FUNCTION_BLOCK FB_HwRefNanotecPD EXTENDS FB_CanNodeBase
VAR_INPUT
	nControlword	AT%Q* : UINT;
	nMode			AT%Q* : SINT;
	nTargetPosition AT%Q* : DINT;
	nTargetSpeed	AT%Q* : INT;
	nDriveSubMode	AT%Q* : UDINT; //1 für Move, 8 für Stillstand mit Stromabsenkung	
END_VAR
VAR_OUTPUT
	nStatusword 	 	AT%I* : UINT;
	nCurrentMode 	 	AT%I* : SINT;
	nCurrentPosition 	AT%I* : DINT;
	nCurrentSpeed		AT%I* : INT;
	nFollowingError		AT%I* : DINT;	
END_VAR
VAR
	bIsHomed 				: BOOL;
	eCurrentSTM				: E_CoDS402States;
	nState 					: USINT;
	bFirstTimeInOperational : BOOL := TRUE;
	
	nStateA_ProcessError	: USINT;
	nLastErrorID			: DWORD;
	nErrorCount				: USINT;
	
	nStateA_ResetError		: USINT;
END_VAR

VAR PERSISTENT
	nDistPerMotorRev	: DINT;
	nRefPos				: DINT;
	nHomePos			: DINT;
	nSlowHomingSpeed	: DINT;
	nFastHomingSpeed	: DINT;
	bInvertInitDir		: BOOL;
	nMinPos				: DINT;
	nMaxPos				: DINT;
	nMaxSpeed			: DINT;
END_VAR

//In der Basisklasse wird A_Prepare und A_ResetApp ausgeführt
//ResetApp ist hier nicht relevant.

eCurrentSTM := M_GetDS402State();
CASE nState OF
	0:	//Prepare
		SUPER^();
		IF bPreparingOK THEN
			nState := 1;
		END_IF
		
	1:	//Operational
		//Wenn hier zum erstem mal hineingesprungen wird, und in error, dann gleich resetten
		IF eCurrentSTM = E_CoDS402States.DS402STATE_Fault OR eCurrentSTM = E_CoDS402States.DS402STATE_FaultReactionActive THEN
			IF bFirstTimeInOperational THEN
				nState := 4;
			ELSE
				nState := 2;
			END_IF
		END_IF
		bFirstTimeInOperational := FALSE;
		
	2:	//Process error
		A_ProcessError();
		IF nStateA_ProcessError = 80 THEN
			//Error auswerten - es werden nur die untersten 16Bit ausgewertet (Error Code siehe Doku NanoTec)
			nLastErrorID := nLastErrorID AND 16#FFFF;
			CASE nLastErrorID OF
				16#1000:	nErrorID := E_ErrorIdHwGeneral.ERRORID_GenericError;
				16#2300:	nErrorID := E_ErrorIdHwGeneral.ERRORID_MotorCurrentExceeded;
				16#3100:	nErrorID := E_ErrorIdHwGeneral.ERRORID_InvalidInputVoltage;
				16#4200:	nErrorID := E_ErrorIdHwGeneral.ERRORID_ControllerTemperature;
				16#5540:	nErrorID := E_ErrorIdHwGeneral.ERRORID_InterlockError;
				16#6010:	nErrorID := E_ErrorIdHwGeneral.ERRORID_SoftwareReset;
				16#6100:	nErrorID := E_ErrorIdHwGeneral.ERRORID_InternalSoftwareError;
				16#6320:	nErrorID := E_ErrorIdHwGeneral.ERRORID_InvalidRatedCurrent;
				16#7113:	nErrorID := E_ErrorIdHwGeneral.ERRORID_BallastResistorOverloaded;
				16#7121:	nErrorID := E_ErrorIdHwGeneral.ERRORID_MotorBlocked;
				16#7200:	nErrorID := E_ErrorIdHwGeneral.ERRORID_InternalError;
				16#7305:	nErrorID := E_ErrorIdHwGeneral.ERRORID_Sensor1Fault;
				16#7306:	nErrorID := E_ErrorIdHwGeneral.ERRORID_Sensor2Fault;
				16#7307:	nErrorID := E_ErrorIdHwGeneral.ERRORID_SensorNFault;
				16#7600:	nErrorID := E_ErrorIdHwGeneral.ERRORID_MemoryError;
				16#8000,16#8100: nErrorID := E_ErrorIdHwGeneral.ERRORID_FieldbusMonitoring;
				16#8130, 16#8200, 16#8210, 16#8220, 16#8240 : nErrorID := E_ErrorIdHwGeneral.ERRORID_CANopenError;	
				16#8400:	nErrorID := E_ErrorIdHwGeneral.ERRORID_SpeedMonitoring;
				16#8611:	nErrorID := E_ErrorIdHwGeneral.ERRORID_FollowingError;
				16#8612:	nErrorID := E_ErrorIdHwGeneral.ERRORID_LimitSwitchExceeded;
			ELSE
				nErrorID := 0;
			END_CASE
			nStateA_ProcessError := 0;
			//Notify error
			stError.HardwareGrp := stHardwareId.eGroup;
			stError.HardwareNr := stHardwareId.nItem;
			stError.POU := E_POU.POU_FB_HwRefNanotecPD;
			stError.POUAction := E_POUACT.POUACT_UNDEFIEND;
			stError.ErrorId := nErrorID;
			fbErrorList.M_Add(stError);
			nState := 3;
		END_IF
		
	3:	//Error
		IF bResetError THEN
			nState:= 4;
			bResetError := FALSE;
		END_IF
		bIsHomed := FALSE;
		bError := TRUE;
		
	4:	//Reset
		bBusy := TRUE;
		A_ResetError();
		IF nStateA_ResetError = 80 THEN
			bError := FALSE;
			bBusy := FALSE;
			nStateA_ResetError := 0;
			nState := 1;
		ELSIF nStateA_ResetError = 99 THEN
			bBusy := FALSE;
			nStateA_ResetError := 0;
			nState := 3;
		END_IF
	
END_CASE

ACTION A_ProcessError:
IF nStateA_ProcessError = 0 THEN
	//Object 0x1003:00 auslesen (Anzahl der Errors im Pre-defined error field)
	fbSdoRead(nIndex:= 16#1003, nSubIndex:= 0, nDataLength:= 1, bExecute:= TRUE);
	nErrorCount := 0;
	IF NOT fbSdoRead.bBusy THEN
		IF NOT fbSdoRead.bError THEN
			nErrorCount := DINT_TO_USINT(fbSdoRead.nData);
		END_IF
		fbSdoRead(bExecute:= FALSE);
		IF nErrorCount > 0 THEN
			nStateA_ProcessError := 1;
		ELSE
			nStateA_ProcessError := 80;
		END_IF
	END_IF
END_IF


IF nStateA_ProcessError = 1 THEN
	//Object 0x1003:01 auslesen (Neuester Error)
	fbSdoRead(nIndex:= 16#1003, nSubIndex:= 1, nDataLength:= 4, bExecute:= TRUE);
	nLastErrorID := 0;
	IF NOT fbSdoRead.bBusy THEN
		IF NOT fbSdoRead.bError THEN
			nLastErrorID := fbSdoRead.nData;
		END_IF
		fbSdoRead(bExecute:= FALSE);
		nStateA_ProcessError := 80;
	END_IF
END_IF
END_ACTION

ACTION A_ResetError:
CASE nStateA_ResetError OF
	0:	
		CASE eCurrentSTM OF
			E_CoDS402States.DS402STATE_Fault:
				nControlword := 153;	//Reset error
			E_CoDS402States.DS402STATE_SwitchOnDisabled:
				nStateA_ResetError := 1;
			E_CoDS402States.DS402STATE_ReadyToSwitchOn:
				nControlword := 0;	//Transition 7 in DS402 statemachine -> geht in Switch on disabled
				nStateA_ResetError := 1;
			E_CoDS402States.DS402STATE_SwitchedOn:
				nControlword := 0;	//Transition 10 in DS402 statemachine -> geht in Switch on disabled
				nStateA_ResetError := 1;
			E_CoDS402States.DS402STATE_OperationEnabled:
				nControlword := 0;	//Shutdown
				nStateA_ResetError := 1;
			E_CoDS402States.DS402STATE_NotReadyToSwitchOn:	//Statusword wahrscheinlich nicht gemappt
				nStateA_ResetError := 99;
		END_CASE
		
	1:	//Würde Antrieb bereits gehomed?
		IF bIsHomed THEN
			nControlword := 6;
			nStateA_ResetError := 2;
		ELSE
			nStateA_ResetError := 80;
		END_IF
		
	2:	IF eCurrentSTM = E_CoDS402States.DS402STATE_ReadyToSwitchOn THEN
			nControlword := 7;	//Change to "Switched on"
			nStateA_ResetError := 3;
		ELSIF eCurrentSTM = E_CoDS402States.DS402STATE_Fault THEN
			nStateA_ResetError := 99;
		END_IF
	
	3:	IF eCurrentSTM = E_CoDS402States.DS402STATE_SwitchedOn THEN
			nControlword := 15;	//Change to "Switched on"
			nStateA_ResetError := 4;
		ELSIF eCurrentSTM = E_CoDS402States.DS402STATE_Fault THEN
			nStateA_ResetError := 99;
		END_IF
		
	4:	IF eCurrentSTM = E_CoDS402States.DS402STATE_OperationEnabled THEN
			nStateA_ResetError := 80;
		ELSIF eCurrentSTM = E_CoDS402States.DS402STATE_Fault THEN
			nStateA_ResetError := 99;
		END_IF		
	
END_CASE
END_ACTION

METHOD M_GetDS402State : E_CoDS402States
VAR_INPUT
END_VAR
IF (nStatusword AND 16#4F) = 0 THEN
	M_GetDS402State := E_CoDS402States.DS402STATE_NotReadyToSwitchOn;
ELSIF (nStatusword AND 16#4F) = 16#40 THEN
	M_GetDS402State := E_CoDS402States.DS402STATE_SwitchOnDisabled;
ELSIF (nStatusword AND 16#6F) = 16#21 THEN
	M_GetDS402State := E_CoDS402States.DS402STATE_ReadyToSwitchOn;
ELSIF (nStatusword AND 16#6F) = 16#23 THEN
	M_GetDS402State := E_CoDS402States.DS402STATE_SwitchedOn;
ELSIF (nStatusword AND 16#6F) = 16#27 THEN
	M_GetDS402State := E_CoDS402States.DS402STATE_OperationEnabled;
ELSIF (nStatusword AND 16#6F) = 16#07 THEN
	M_GetDS402State := E_CoDS402States.DS402STATE_QuickStopActive;
ELSIF (nStatusword AND 16#4F) = 16#0F THEN
	M_GetDS402State := E_CoDS402States.DS402STATE_FaultReactionActive;
ELSIF (nStatusword AND 16#4F) = 16#08 THEN
	M_GetDS402State := E_CoDS402States.DS402STATE_Fault;
ELSE
	M_GetDS402State := E_CoDS402States.DS402STATE_Notspecified;
END_IF
END_METHOD

METHOD M_GetHomingState : E_CoDS402HomingState
VAR_INPUT
END_VAR

VAR 
END_VAR
//werted nur die Bits 10,12,13 vom Statusword aus
CASE nStatusword AND 16#3400 OF
	16#0000:	M_GetHomingState := E_CoDS402HomingState.HomingInProgress;
	16#0400:	M_GetHomingState := E_CoDS402HomingState.HomingInteruptedOrNotReached;
	16#1000:	M_GetHomingState := E_CoDS402HomingState.HomingAttainedButNotReached;
	16#1400:	M_GetHomingState := E_CoDS402HomingState.HomingSuccess;
	16#2000,
	16#2400		:M_GetHomingState := E_CoDS402HomingState.HomingError;
END_CASE
END_METHOD

METHOD M_RealToInternPos : DINT
VAR_INPUT
	nValue : DINT;
END_VAR
M_RealToInternPos := REAL_TO_DINT(DINT_TO_REAL(nValue) * 2000.0 / DINT_TO_REAL(nDistPerMotorRev));
END_METHOD

METHOD M_RealToInternSpeed : INT
VAR_INPUT
	nValue : DINT; //Speed in µm/s oder 1/100°/sec
END_VAR
//Umrechnung in U/min
M_RealToInternSpeed := REAL_TO_INT(DINT_TO_REAL(nValue) / DINT_TO_REAL(nDistPerMotorRev) * 60.0);
RETURN;
END_METHOD

METHOD M_SetTargetPos : BOOL
VAR_INPUT
	nValue : DINT; //Reale Einheit
END_VAR
IF (nValue >= nMinPos) AND (nValue <= nMaxPos) THEN
	nTargetPosition :=  REAL_TO_DINT(DINT_TO_REAL(nValue) * 2000.0 / DINT_TO_REAL(nDistPerMotorRev));
	M_SetTargetPos := TRUE;
END_IF
END_METHOD

METHOD M_SetTargetSpeed : BOOL
VAR_INPUT
	nValue : DINT; //Reale Einheit
END_VAR
IF (nValue >= 0) AND (nValue <= nMaxSpeed) THEN
	nTargetSpeed := M_RealToInternSpeed(nValue);
	M_SetTargetSpeed := TRUE;
END_IF
END_METHOD

PROPERTY P_bInvertInitDir : BOOL
GET
P_bInvertInitDir := bInvertInitDir;
END_GET
SET
bInvertInitDir := P_bInvertInitDir;
fbSettings.M_WritePersData();
END_SET
END_PROPERTY

PROPERTY P_bIsHomed : BOOL
GET
P_bIsHomed := bIsHomed;
END_GET
SET
bIsHomed := P_bIsHomed;
END_SET
END_PROPERTY

PROPERTY P_nCurrentRealPos : DINT
GET
P_nCurrentRealPos := REAL_TO_DINT(DINT_TO_REAL(nCurrentPosition) / 2000.0 * DINT_TO_REAL(nDistPerMotorRev));
END_GET
END_PROPERTY

PROPERTY P_nDistPerMotorRev : DINT
GET
P_nDistPerMotorRev := nDistPerMotorRev;
END_GET
SET
nDistPerMotorRev := P_nDistPerMotorRev;
fbSettings.M_WritePersData();
END_SET
END_PROPERTY

PROPERTY P_nErrorID : ERRORID
GET
P_nErrorID := nErrorId;
END_GET
END_PROPERTY

PROPERTY P_nFastHomingSpeed : DINT
GET
P_nFastHomingSpeed := nFastHomingSpeed;
END_GET
SET
nFastHomingSpeed := P_nFastHomingSpeed;
fbSettings.M_WritePersData();
END_SET
END_PROPERTY

PROPERTY P_nHomePos : DINT
GET
P_nHomePos := nHomePos;
END_GET
SET
nHomePos := P_nHomePos;
fbSettings.M_WritePersData();
END_SET
END_PROPERTY

PROPERTY P_nMaxPos : DINT
GET
P_nMaxPos := nMaxPos;
END_GET
SET
nMaxPos := P_nMaxPos;
fbSettings.M_WritePersData();
END_SET
END_PROPERTY

PROPERTY P_nMaxSpeed : DINT
GET
P_nMaxSpeed := nMaxSpeed;
END_GET
SET
nMaxSpeed := P_nMaxSpeed;
fbSettings.M_WritePersData();
END_SET
END_PROPERTY

PROPERTY P_nMinPos : DINT
GET
P_nMinPos := nMinPos;
END_GET
SET
nMinPos := P_nMinPos;
fbSettings.M_WritePersData();
END_SET
END_PROPERTY

PROPERTY P_nRefPos : DINT
GET
P_nRefPos := nRefPos;
END_GET
SET
nRefPos := P_nRefPos;
fbSettings.M_WritePersData();
END_SET
END_PROPERTY

PROPERTY P_nSlowHomingSpeed : DINT
GET
P_nSlowHomingSpeed := nSlowHomingSpeed;
END_GET
SET
nSlowHomingSpeed := P_nSlowHomingSpeed;
fbSettings.M_WritePersData();
END_SET
END_PROPERTY

END_FUNCTION_BLOCK

(* stored: Version 1.1.0.1, ProductVersion 3.1.4024.11
   POU FB_HwRefNanotecPD: Id {66629387-bdd7-4093-89b1-13f9ee2856fa}, SpecialFunc None
   Action A_ProcessError: Id {202f49b2-ecc0-45fe-93e8-7f8c6b182e23}
   Action A_ResetError: Id {2ad7e5dc-046a-44f3-9de9-b310f5a0f7e8}
   Method M_GetDS402State: Id {d35cebfa-d2cf-4fa6-8922-06e262aa7052}
   Method M_GetHomingState: Id {2fd3c8d8-056d-4234-8f2b-93aa7e91d53f}
   Method M_RealToInternPos: Id {6edadc39-af5b-4a72-aa2a-31f930f31d57}
   Method M_RealToInternSpeed: Id {8d587905-06e7-4735-b77d-d09846d59df8}
   Method M_SetTargetPos: Id {9616795f-cabd-4830-8f7e-f3e6344cca2d}
   Method M_SetTargetSpeed: Id {50cbe063-7bd5-47b1-b264-aa1a8b37aab9}
   Property P_bInvertInitDir: Id {8c47b135-2bba-4c39-b0fd-843d77dac176}
   Get Get: Id {1fef854f-142c-493c-9d1b-6766b13a402c}
   Set Set: Id {2f50b62c-d963-4157-ac19-d09495717ecc}
   Property P_bIsHomed: Id {4456ecb3-c12b-47c1-9bc2-c0e8a6628615}
   Get Get: Id {66004908-3c1b-4458-83e7-3236decbe45f}
   Set Set: Id {32512070-f624-44d7-9d96-5ae7212d7fd9}
   Property P_nCurrentRealPos: Id {c92a3468-c1c3-4a90-b561-52343f71e77e}
   Get Get: Id {184fcefd-66a0-4775-9f09-b6359bba7578}
   Property P_nDistPerMotorRev: Id {15d9a758-9564-489b-ae12-651dae792d45}
   Get Get: Id {78374e61-8a80-40ee-9139-dab59fabfbdc}
   Set Set: Id {3c66ebe1-a82b-40b5-82e8-1d45ffe5f4c2}
   Property P_nErrorID: Id {cba448cf-3331-41f4-8a3f-0db767dae882}
   Get Get: Id {ae27c062-6a23-4308-8b67-19d2f9fefdcc}
   Property P_nFastHomingSpeed: Id {02368013-d887-4cd6-8eb0-01e67ece8af2}
   Get Get: Id {3db5a4f2-bf6a-41a0-a3fa-9e8809c7852c}
   Set Set: Id {20a14a4b-bf90-43eb-b27a-b449ecd23292}
   Property P_nHomePos: Id {f6960b24-6899-4908-ac51-e85760b5b39d}
   Get Get: Id {5fe98fc1-6b5b-4e35-98c1-3823d8e68e30}
   Set Set: Id {59f66c91-7239-48cd-b01a-88080e7c0378}
   Property P_nMaxPos: Id {5e9a9c09-829e-46f5-b4ef-d42ad64ef519}
   Get Get: Id {4f20f08b-3168-40f0-bd74-7273b896af8b}
   Set Set: Id {07a8d019-57fe-49d1-800d-d277e539f2e4}
   Property P_nMaxSpeed: Id {79b3c601-3251-43d5-a1f8-34754eba39fb}
   Get Get: Id {e92051a9-2e62-4ac9-80a2-3459e56260e4}
   Set Set: Id {2e41349c-e1e5-4858-9124-a70d5fdd1544}
   Property P_nMinPos: Id {578b2cf2-5df8-4e8e-8176-da29f6ad3d84}
   Get Get: Id {aa6ccf19-fa48-40fb-80c3-a811de061025}
   Set Set: Id {20d3fad0-6b06-401c-b832-06a676f2ac45}
   Property P_nRefPos: Id {75f154d2-e22c-4ec1-9f4e-8d4723bf492b}
   Get Get: Id {b1312a12-7834-4130-a109-a476e63b9092}
   Set Set: Id {02697c0b-04a4-49eb-b475-35c2db0ee1a9}
   Property P_nSlowHomingSpeed: Id {827a7fb9-f535-4e2a-90ab-1a5b7876b87b}
   Get Get: Id {606b688f-0c26-4ffc-a715-299457198b34}
   Set Set: Id {97da0881-7f9f-40c6-8362-0c589da44b57} *)
